{attribute addProperty BoxType "EJ1819-0000-0017"}
{attribute addProperty Id "ChannelAT %I*ARRAY[0..15] OF Channel_E4AEF59E128160WcStateAT %I*WcState_98A4DF7520.250InfoDataAT %I*InfoData_192954DE1620"}
{attribute addProperty CRC "4206052659"}
{attribute addProperty SizeInBites "146"}
{attribute addProperty SizeInBytes "18.25"}
TYPE EJ1819_248EAA34 :
STRUCT
	{attribute addProperty Name "Channel"}
	Channel : ARRAY[0..15] OF Channel_E4AEF59E;
	{attribute addProperty Name "WcState"}
	WcState : WcState_98A4DF75;
	{attribute addProperty Name "InfoData"}
	InfoData : InfoData_192954DE;
END_STRUCT
END_TYPE

(* stored: Version 1.2.0.0, ProductVersion 3.1.4024.9
   DUT EJ1819_248EAA34: Id {b1a47d40-af7d-4497-81aa-0f774e2d7f85} *)
